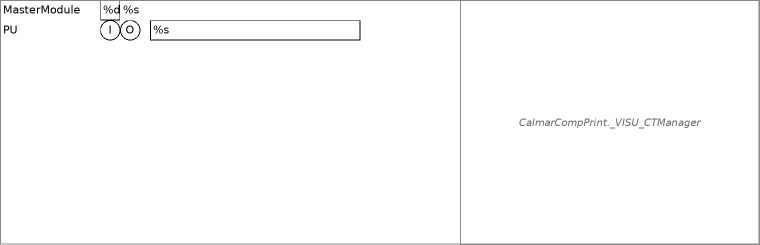
VISUALIZATION _VISU_ModuleMaster  // 760x245
VAR_IN_OUT
	mInst : FB_ModuleMaster;
END_VAR
    Rectangle (150,20 210x20), "%s", tooltip "%s", text variable: mInst._pPU^._activeJob^._sActiveJobDef.sJobSettings.aI_JobName, colour toggle: mInst._pPU^._activeJob <> 0
        p4168582468: mInst._pPU^._activeJob^._sActiveJobDef.sJobSettings.aI_JobName
    Ellipse (100,20 20x20), "I", colour toggle: mInst._pPU^._pAdsPu^.sI_Start.bI_Command OR mInst._pPU^._pAdsPu^.sI_Start.bO_CommandCanEx
        tap mInst._pPU^._pAdsPu^.sI_Start.bI_Command
    Ellipse (120,20 20x20), "O", colour toggle: mInst._pPU^._pAdsPu^.sI_Stop.bI_Command OR mInst._pPU^._pAdsPu^.sI_Stop.bO_CommandCanEx
        tap mInst._pPU^._pAdsPu^.sI_Stop.bI_Command
    Rectangle (100,0 20x20), "%d", tooltip "Master module idx", text variable: mInst._pMasterModule^._nIdx
    Rectangle (0,0 100x20), "MasterModule"
    Rectangle (0,20 100x20), "PU"
    Rectangle (120,0 240x20), "%s", text variable: mInst._pMasterModule^._instanceName
    Frame (460,0 300x245)
        shows CalmarCompPrint._VISU_CTManager(m_Inst := mInst.fBCTManagerMain)
END_VISUALIZATION

(* stored: Version 1.1.0.1, ProductVersion 3.1.4024.11
   Visu _VISU_ModuleMaster: Id {c1d8c7a3-7d0d-4a3b-9a26-2906f1530475} *)
